TYPE ST_DB_Record :
STRUCT

Float1	:	LREAL;
Float2	:	LREAL;	
Float3	:	LREAL;
Float4	:	LREAL;	
Float5	:	LREAL;


END_STRUCT
END_TYPE

(* stored: Version 1.1.0.1, ProductVersion 3.1.4022.18
   DUT ST_DB_Record: Id {045fff51-b2a7-4e42-a929-5966d063d9db} *)
